// TIA Portal V15.1 export
// export: Created 2024-06-21T08:41:00.5751261Z, ExportSetting WithDefaults, DisplayName Totally Integrated Automation Portal, DisplayVersion V15.1 Update 5, DisplayName TIA Portal Openness, DisplayVersion V15.1 Update 5, DisplayName SINAMICS Startdrive Advanced, DisplayVersion V15.1, DisplayName G130, G150, S120, S150, SINAMICS MV, S210, DisplayVersion V15.1, DisplayName G110M, G120, G120C, G120D, G120P, DisplayVersion V15.1, DisplayName STEP 7 Professional, DisplayVersion V15.1 Update 5, DisplayName STEP 7 Safety, DisplayVersion V15.1, DisplayName WinCC Professional, DisplayVersion V15.1 Update 5, DisplayName SIMATIC Visualization Architect, DisplayVersion V15.1
FUNCTION_BLOCK "LMDBToDB"   // FB2145, FBD
TITLE = LMDBToDB
{ S7_Optimized_Access := 'FALSE' }
AUTHOR : VCC
FAMILY : DataHand
VERSION : 0.1
// =============================================================================
// This module Copies data from DB to DB
// =============================================================================
// stored: AutoNumber false, IsIECCheckEnabled true, SetENOAutomatically False, UDAEnableTagReadback false
   VAR_INPUT
      I_CopyDB { ExternalAccessible := 'False'; ExternalVisible := 'False'; ExternalWritable := 'False'} : Bool;   // Copy DB
      I_SourceDB { ExternalAccessible := 'False'; ExternalVisible := 'False'; ExternalWritable := 'False'} : DB_ANY;   // Source DB
      I_StartAddresSourceDB { ExternalAccessible := 'False'; ExternalVisible := 'False'; ExternalWritable := 'False'} : Int;   // Address
      I_DestDB { ExternalAccessible := 'False'; ExternalVisible := 'False'; ExternalWritable := 'False'} : DB_ANY;   // Dest DB
      I_StartAddressDestDB { ExternalAccessible := 'False'; ExternalVisible := 'False'; ExternalWritable := 'False'} : Int;   // Address
      I_LenghtBytes { ExternalAccessible := 'False'; ExternalVisible := 'False'; ExternalWritable := 'False'} : Word;   // Length
   END_VAR
   VAR_TEMP
      SourcePointer : Any;   // Temp
      DestPointer : Any;   // Temp
      SourceDB : Int;   // Temp
      DestDB : Int;   // Temp
   END_VAR
BEGIN

NETWORK
TITLE = **** 1 - Inputs **** DB Pointers
// DB Pointers
      OPN   #I_SourceDB;
      L     DBNO;
      T     #SourceDB;
      OPN   #I_DestDB;
      L     DBNO;
      T     #DestDB;

NETWORK
TITLE = **** 5.2 - Equations - Flow Equations **** Load Pointers
// Load Pointers
// APa Cleaning Warnings
      A     #I_CopyDB;
      JCN   ncAp;
      LAR1  P##SourcePointer;
      L     16#1002;
      T     LW [AR1, P#0.0];
      L     #I_LenghtBytes;
      T     LW [AR1, P#2.0];
      L     #SourceDB;
      T     LW [AR1, P#4.0];
      L     #I_StartAddresSourceDB;
      SLD   3;
      OD    16#8400_0000;
      T     LD [AR1, P#6.0];
      LAR1  P##DestPointer;
      L     16#1002;
      T     LW [AR1, P#0.0];
      L     #I_LenghtBytes;
      T     LW [AR1, P#2.0];
      L     #DestDB;
      T     LW [AR1, P#4.0];
      L     #I_StartAddressDestDB;
      SLD   3;
      OD    16#8400_0000;
      T     LD [AR1, P#6.0];
//      L     16#1002
//      T     %LW10
//      L     #I_LenghtBytes
//      T     %LW12
//      L     #DestDB
//      T     %LW14
//      L     #I_StartAddressDestDB
//      SLD   3
//      OD    16#8400_0000
//      T     %LD16
      CALL  BLKMOV
      ( SRCBLK  := #SourcePointer,
        RET_VAL := "NotUsedInt",
        DSTBLK  := #DestPointer
      );
ncAp: NOP   0;
END_FUNCTION_BLOCK
